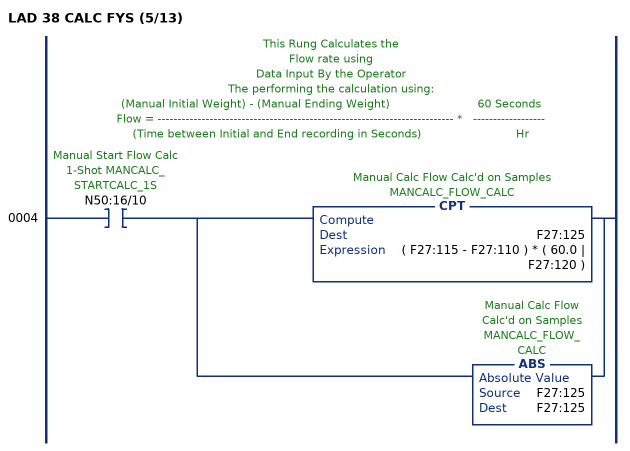
% Rung: 4 %
% This Rung Calculates the
% Flow rate using
% Data Input By the Operator
% The performing the calculation using:
% 
%              (Manual Initial Weight) - (Manual Ending Weight)                         60 Seconds
% Flow = -------------------------------------------------------------------------- *   ------------------
%    (Time between Initial and End recording in Seconds)                           Hr %
SOR XIC N50:16/10 BST CPT F27:125 " ( F27:115 - F27:110 ) * ( 60.0 | F27:120 ) " NXB ABS F27:125 F27:125 BND EOR
%   N50:16/10  MANCALC_STARTCALC_1S  "Manual Start Flow Calc 1-Shot" %
%   F27:125  MANCALC_FLOW_CALC  "Manual Calc Flow Calc'd on Samples" %
%   F27:115  MANCALC_END_VALUE  "Manual Calc End Value for Flow Calc (Lb's)" %
%   F27:110  MANCALC_INIT_VALUE  "Manual Calc Initial Value for Flow Calc (Lb's)" %
%   F27:120  MANCALC_TIME  "Manual Calc Time for Flow Calc (Min's)" %

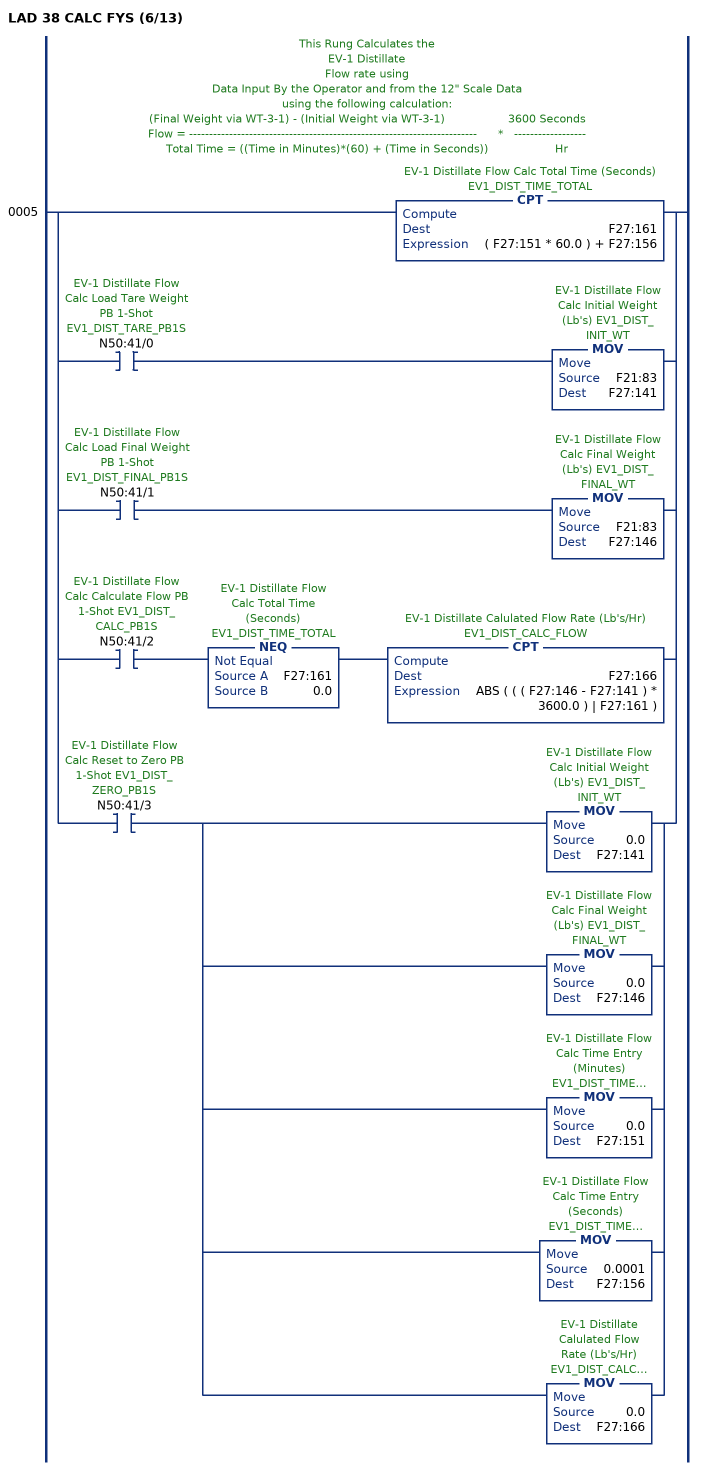
% Rung: 5 %
% This Rung Calculates the
% EV-1 Distillate
% Flow rate using
% Data Input By the Operator and from the 12" Scale Data
% using the following calculation:
% 
%              (Final Weight via WT-3-1) - (Initial Weight via WT-3-1)                  3600 Seconds
% Flow = ------------------------------------------------------------------------      *   ------------------
%    Total Time = ((Time in Minutes)*(60) + (Time in Seconds))                   Hr %
SOR BST CPT F27:161 " ( F27:151 * 60.0 ) + F27:156 " NXB XIC N50:41/0 MOV F21:83 F27:141 NXB XIC N50:41/1 MOV F21:83 F27:146 NXB XIC N50:41/2 NEQ F27:161 0.0 CPT F27:166 " ABS ( ( ( F27:146 - F27:141 ) * 3600.0 ) | F27:161 ) " NXB XIC N50:41/3 BST MOV 0.0 F27:141 NXB MOV 0.0 F27:146 NXB MOV 0.0 F27:151 NXB MOV 0.0001 F27:156 NXB MOV 0.0 F27:166 BND BND EOR
%   F27:161  EV1_DIST_TIME_TOTAL  "EV-1 Distillate Flow Calc Total Time (Seconds)" %
%   F27:151  EV1_DIST_TIME_MINS  "EV-1 Distillate Flow Calc Time Entry (Minutes)" %
%   F27:156  EV1_DIST_TIME_SECS  "EV-1 Distillate Flow Calc Time Entry (Seconds)" %
%   N50:41/0  EV1_DIST_TARE_PB1S  "EV-1 Distillate Flow Calc Load Tare Weight PB 1-Shot" %
%   F21:83  WY0301  "WY-3-1 Platform Scale No-3 Weight 12" x 12" Scale" %
%   F27:141  EV1_DIST_INIT_WT  "EV-1 Distillate Flow Calc Initial Weight (Lb's)" %
%   N50:41/1  EV1_DIST_FINAL_PB1S  "EV-1 Distillate Flow Calc Load Final Weight PB 1-Shot" %
%   F27:146  EV1_DIST_FINAL_WT  "EV-1 Distillate Flow Calc Final Weight (Lb's)" %
%   N50:41/2  EV1_DIST_CALC_PB1S  "EV-1 Distillate Flow Calc Calculate Flow PB 1-Shot" %
%   F27:166  EV1_DIST_CALC_FLOW  "EV-1 Distillate Calulated Flow Rate (Lb's/Hr)" %
%   N50:41/3  EV1_DIST_ZERO_PB1S  "EV-1 Distillate Flow Calc Reset to Zero PB 1-Shot" %

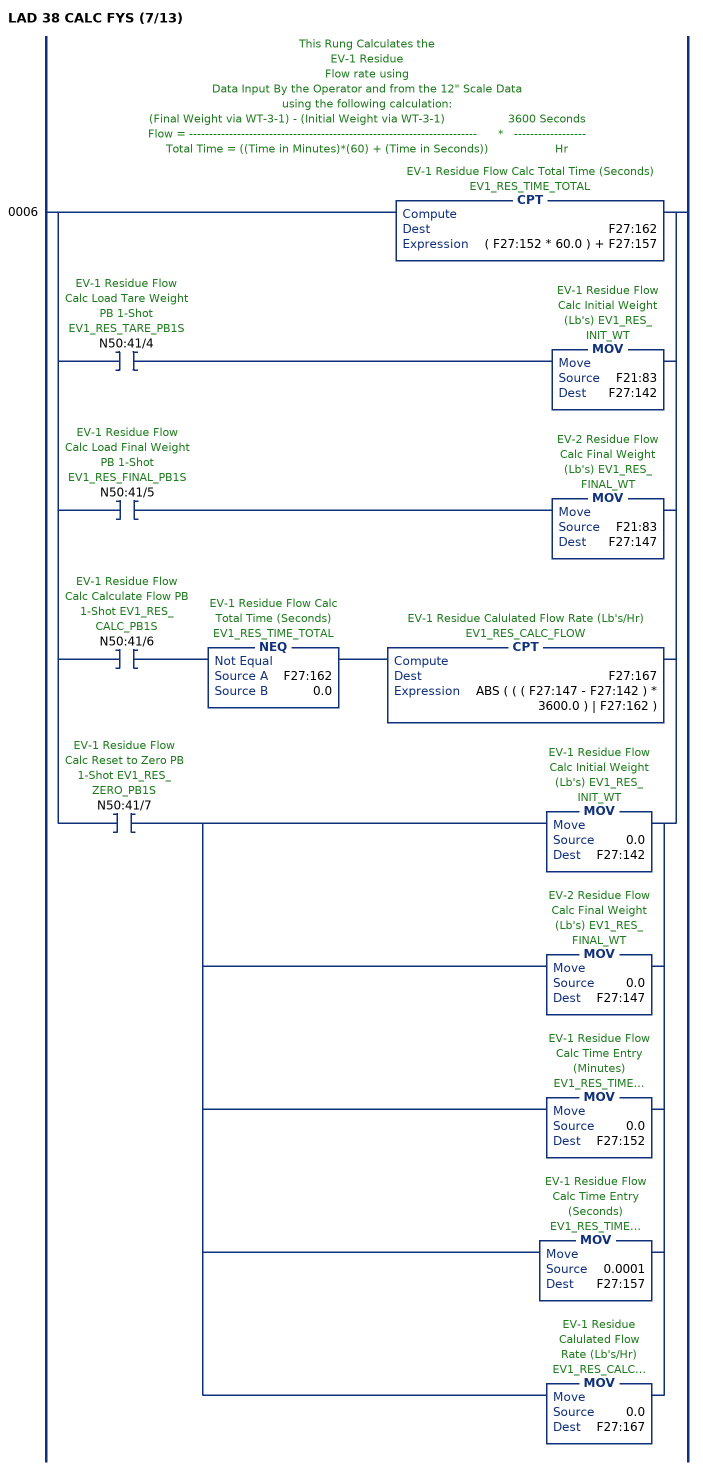
% Rung: 6 %
% This Rung Calculates the
% EV-1 Residue
% Flow rate using
% Data Input By the Operator and from the 12" Scale Data
% using the following calculation:
% 
%              (Final Weight via WT-3-1) - (Initial Weight via WT-3-1)                  3600 Seconds
% Flow = ------------------------------------------------------------------------      *   ------------------
%    Total Time = ((Time in Minutes)*(60) + (Time in Seconds))                   Hr %
SOR BST CPT F27:162 " ( F27:152 * 60.0 ) + F27:157 " NXB XIC N50:41/4 MOV F21:83 F27:142 NXB XIC N50:41/5 MOV F21:83 F27:147 NXB XIC N50:41/6 NEQ F27:162 0.0 CPT F27:167 " ABS ( ( ( F27:147 - F27:142 ) * 3600.0 ) | F27:162 ) " NXB XIC N50:41/7 BST MOV 0.0 F27:142 NXB MOV 0.0 F27:147 NXB MOV 0.0 F27:152 NXB MOV 0.0001 F27:157 NXB MOV 0.0 F27:167 BND BND EOR
%   F27:162  EV1_RES_TIME_TOTAL  "EV-1 Residue Flow Calc Total Time (Seconds)" %
%   F27:152  EV1_RES_TIME_MINS  "EV-1 Residue Flow Calc Time Entry (Minutes)" %
%   F27:157  EV1_RES_TIME_SECS  "EV-1 Residue Flow Calc Time Entry (Seconds)" %
%   N50:41/4  EV1_RES_TARE_PB1S  "EV-1 Residue Flow Calc Load Tare Weight PB 1-Shot" %
%   F21:83  WY0301  "WY-3-1 Platform Scale No-3 Weight 12" x 12" Scale" %
%   F27:142  EV1_RES_INIT_WT  "EV-1 Residue Flow Calc Initial Weight (Lb's)" %
%   N50:41/5  EV1_RES_FINAL_PB1S  "EV-1 Residue Flow Calc Load Final Weight PB 1-Shot" %
%   F27:147  EV1_RES_FINAL_WT  "EV-2 Residue Flow Calc Final Weight (Lb's)" %
%   N50:41/6  EV1_RES_CALC_PB1S  "EV-1 Residue Flow Calc Calculate Flow PB 1-Shot" %
%   F27:167  EV1_RES_CALC_FLOW  "EV-1 Residue Calulated Flow Rate (Lb's/Hr)" %
%   N50:41/7  EV1_RES_ZERO_PB1S  "EV-1 Residue Flow Calc Reset to Zero PB 1-Shot" %

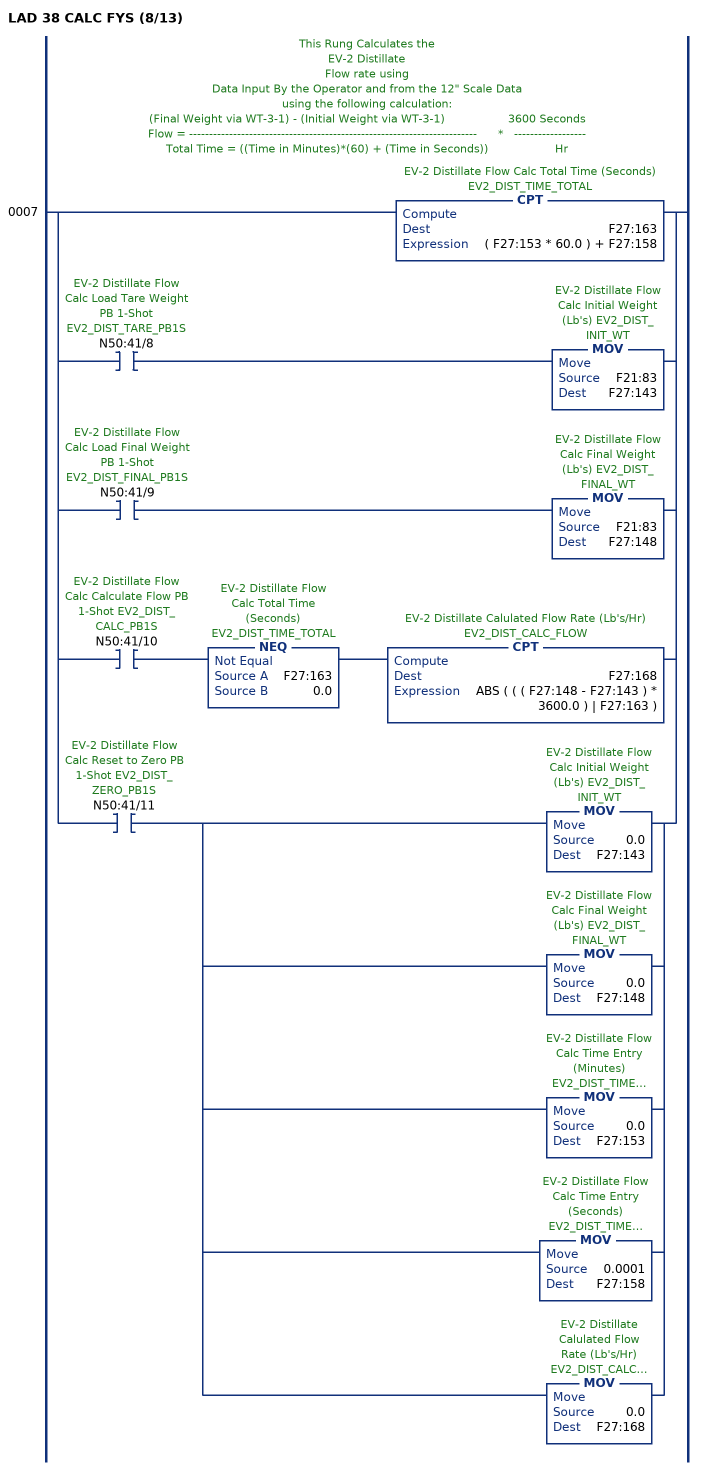
% Rung: 7 %
% This Rung Calculates the
% EV-2 Distillate
% Flow rate using
% Data Input By the Operator and from the 12" Scale Data
% using the following calculation:
% 
%              (Final Weight via WT-3-1) - (Initial Weight via WT-3-1)                  3600 Seconds
% Flow = ------------------------------------------------------------------------      *   ------------------
%    Total Time = ((Time in Minutes)*(60) + (Time in Seconds))                   Hr %
SOR BST CPT F27:163 " ( F27:153 * 60.0 ) + F27:158 " NXB XIC N50:41/8 MOV F21:83 F27:143 NXB XIC N50:41/9 MOV F21:83 F27:148 NXB XIC N50:41/10 NEQ F27:163 0.0 CPT F27:168 " ABS ( ( ( F27:148 - F27:143 ) * 3600.0 ) | F27:163 ) " NXB XIC N50:41/11 BST MOV 0.0 F27:143 NXB MOV 0.0 F27:148 NXB MOV 0.0 F27:153 NXB MOV 0.0001 F27:158 NXB MOV 0.0 F27:168 BND BND EOR
%   F27:163  EV2_DIST_TIME_TOTAL  "EV-2 Distillate Flow Calc Total Time (Seconds)" %
%   F27:153  EV2_DIST_TIME_MINS  "EV-2 Distillate Flow Calc Time Entry (Minutes)" %
%   F27:158  EV2_DIST_TIME_SECS  "EV-2 Distillate Flow Calc Time Entry (Seconds)" %
%   N50:41/8  EV2_DIST_TARE_PB1S  "EV-2 Distillate Flow Calc Load Tare Weight PB 1-Shot" %
%   F21:83  WY0301  "WY-3-1 Platform Scale No-3 Weight 12" x 12" Scale" %
%   F27:143  EV2_DIST_INIT_WT  "EV-2 Distillate Flow Calc Initial Weight (Lb's)" %
%   N50:41/9  EV2_DIST_FINAL_PB1S  "EV-2 Distillate Flow Calc Load Final Weight PB 1-Shot" %
%   F27:148  EV2_DIST_FINAL_WT  "EV-2 Distillate Flow Calc Final Weight (Lb's)" %
%   N50:41/10  EV2_DIST_CALC_PB1S  "EV-2 Distillate Flow Calc Calculate Flow PB 1-Shot" %
%   F27:168  EV2_DIST_CALC_FLOW  "EV-2 Distillate Calulated Flow Rate (Lb's/Hr)" %
%   N50:41/11  EV2_DIST_ZERO_PB1S  "EV-2 Distillate Flow Calc Reset to Zero PB 1-Shot" %

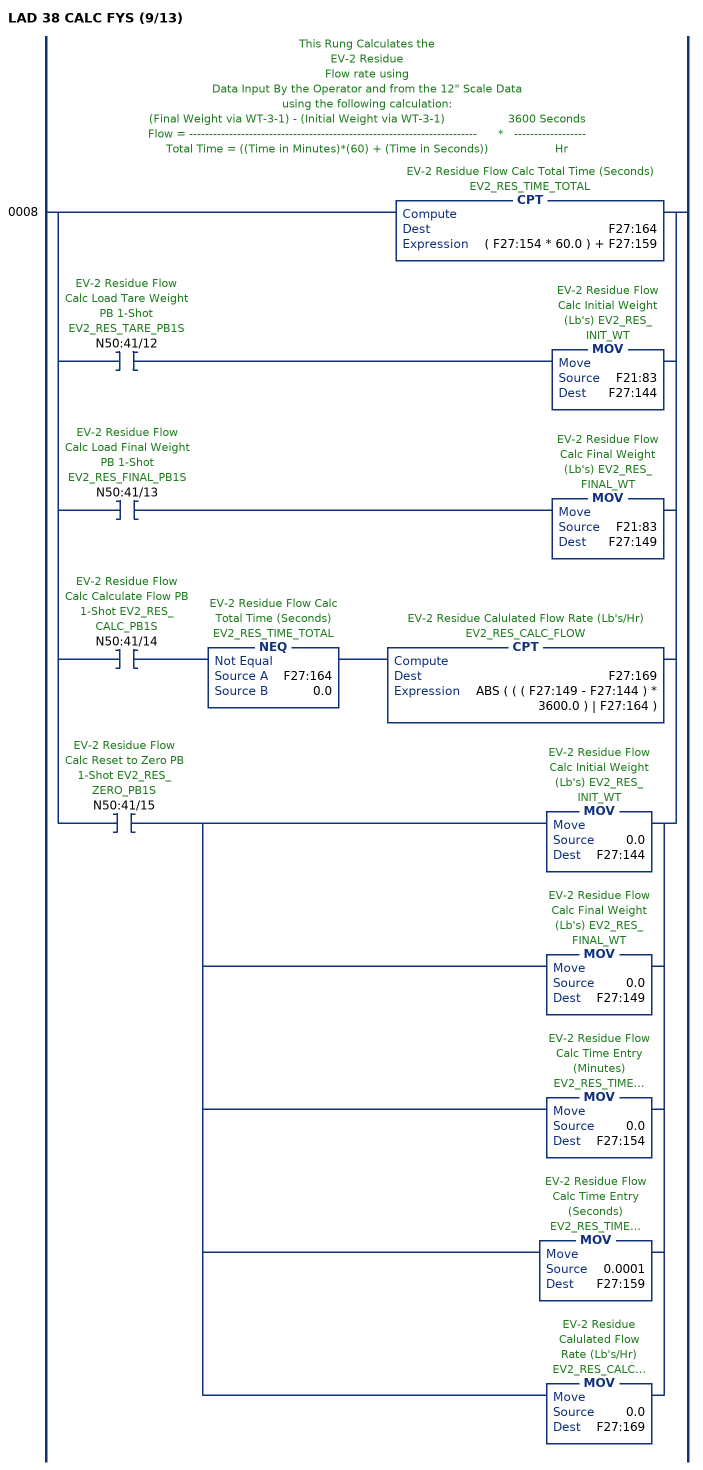
% Rung: 8 %
% This Rung Calculates the
% EV-2 Residue
% Flow rate using
% Data Input By the Operator and from the 12" Scale Data
% using the following calculation:
% 
%              (Final Weight via WT-3-1) - (Initial Weight via WT-3-1)                  3600 Seconds
% Flow = ------------------------------------------------------------------------      *   ------------------
%    Total Time = ((Time in Minutes)*(60) + (Time in Seconds))                   Hr %
SOR BST CPT F27:164 " ( F27:154 * 60.0 ) + F27:159 " NXB XIC N50:41/12 MOV F21:83 F27:144 NXB XIC N50:41/13 MOV F21:83 F27:149 NXB XIC N50:41/14 NEQ F27:164 0.0 CPT F27:169 " ABS ( ( ( F27:149 - F27:144 ) * 3600.0 ) | F27:164 ) " NXB XIC N50:41/15 BST MOV 0.0 F27:144 NXB MOV 0.0 F27:149 NXB MOV 0.0 F27:154 NXB MOV 0.0001 F27:159 NXB MOV 0.0 F27:169 BND BND EOR
%   F27:164  EV2_RES_TIME_TOTAL  "EV-2 Residue Flow Calc Total Time (Seconds)" %
%   F27:154  EV2_RES_TIME_MINS  "EV-2 Residue Flow Calc Time Entry (Minutes)" %
%   F27:159  EV2_RES_TIME_SECS  "EV-2 Residue Flow Calc Time Entry (Seconds)" %
%   N50:41/12  EV2_RES_TARE_PB1S  "EV-2 Residue Flow Calc Load Tare Weight PB 1-Shot" %
%   F21:83  WY0301  "WY-3-1 Platform Scale No-3 Weight 12" x 12" Scale" %
%   F27:144  EV2_RES_INIT_WT  "EV-2 Residue Flow Calc Initial Weight (Lb's)" %
%   N50:41/13  EV2_RES_FINAL_PB1S  "EV-2 Residue Flow Calc Load Final Weight PB 1-Shot" %
%   F27:149  EV2_RES_FINAL_WT  "EV-2 Residue Flow Calc Final Weight (Lb's)" %
%   N50:41/14  EV2_RES_CALC_PB1S  "EV-2 Residue Flow Calc Calculate Flow PB 1-Shot" %
%   F27:169  EV2_RES_CALC_FLOW  "EV-2 Residue Calulated Flow Rate (Lb's/Hr)" %
%   N50:41/15  EV2_RES_ZERO_PB1S  "EV-2 Residue Flow Calc Reset to Zero PB 1-Shot" %

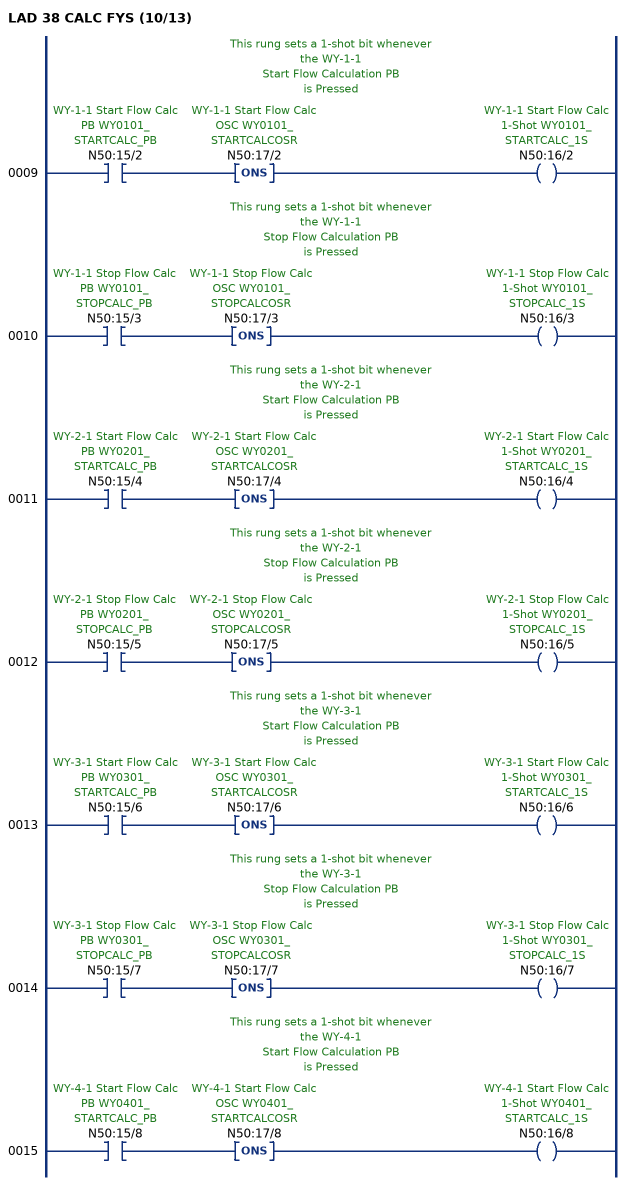
% Rung: 9 %
% This rung sets a 1-shot bit whenever
% the WY-1-1
% Start Flow Calculation PB
% is Pressed %
SOR XIC N50:15/2 OSR N50:17/2 OTE N50:16/2 EOR
%   N50:15/2  WY0101_STARTCALC_PB  "WY-1-1 Start Flow Calc PB" %
%   N50:17/2  WY0101_STARTCALCOSR  "WY-1-1 Start Flow Calc OSC" %
%   N50:16/2  WY0101_STARTCALC_1S  "WY-1-1 Start Flow Calc 1-Shot" %
% Rung: 10 %
% This rung sets a 1-shot bit whenever
% the WY-1-1
% Stop Flow Calculation PB
% is Pressed %
SOR XIC N50:15/3 OSR N50:17/3 OTE N50:16/3 EOR
%   N50:15/3  WY0101_STOPCALC_PB  "WY-1-1 Stop Flow Calc PB" %
%   N50:17/3  WY0101_STOPCALCOSR  "WY-1-1 Stop Flow Calc OSC" %
%   N50:16/3  WY0101_STOPCALC_1S  "WY-1-1 Stop Flow Calc 1-Shot" %
% Rung: 11 %
% This rung sets a 1-shot bit whenever
% the WY-2-1
% Start Flow Calculation PB
% is Pressed %
SOR XIC N50:15/4 OSR N50:17/4 OTE N50:16/4 EOR
%   N50:15/4  WY0201_STARTCALC_PB  "WY-2-1 Start Flow Calc PB" %
%   N50:17/4  WY0201_STARTCALCOSR  "WY-2-1 Start Flow Calc OSC" %
%   N50:16/4  WY0201_STARTCALC_1S  "WY-2-1 Start Flow Calc 1-Shot" %
% Rung: 12 %
% This rung sets a 1-shot bit whenever
% the WY-2-1
% Stop Flow Calculation PB
% is Pressed %
SOR XIC N50:15/5 OSR N50:17/5 OTE N50:16/5 EOR
%   N50:15/5  WY0201_STOPCALC_PB  "WY-2-1 Stop Flow Calc PB" %
%   N50:17/5  WY0201_STOPCALCOSR  "WY-2-1 Stop Flow Calc OSC" %
%   N50:16/5  WY0201_STOPCALC_1S  "WY-2-1 Stop Flow Calc 1-Shot" %
% Rung: 13 %
% This rung sets a 1-shot bit whenever
% the WY-3-1
% Start Flow Calculation PB
% is Pressed %
SOR XIC N50:15/6 OSR N50:17/6 OTE N50:16/6 EOR
%   N50:15/6  WY0301_STARTCALC_PB  "WY-3-1 Start Flow Calc PB" %
%   N50:17/6  WY0301_STARTCALCOSR  "WY-3-1 Start Flow Calc OSC" %
%   N50:16/6  WY0301_STARTCALC_1S  "WY-3-1 Start Flow Calc 1-Shot" %
% Rung: 14 %
% This rung sets a 1-shot bit whenever
% the WY-3-1
% Stop Flow Calculation PB
% is Pressed %
SOR XIC N50:15/7 OSR N50:17/7 OTE N50:16/7 EOR
%   N50:15/7  WY0301_STOPCALC_PB  "WY-3-1 Stop Flow Calc PB" %
%   N50:17/7  WY0301_STOPCALCOSR  "WY-3-1 Stop Flow Calc OSC" %
%   N50:16/7  WY0301_STOPCALC_1S  "WY-3-1 Stop Flow Calc 1-Shot" %
% Rung: 15 %
% This rung sets a 1-shot bit whenever
% the WY-4-1
% Start Flow Calculation PB
% is Pressed %
SOR XIC N50:15/8 OSR N50:17/8 OTE N50:16/8 EOR
%   N50:15/8  WY0401_STARTCALC_PB  "WY-4-1 Start Flow Calc PB" %
%   N50:17/8  WY0401_STARTCALCOSR  "WY-4-1 Start Flow Calc OSC" %
%   N50:16/8  WY0401_STARTCALC_1S  "WY-4-1 Start Flow Calc 1-Shot" %

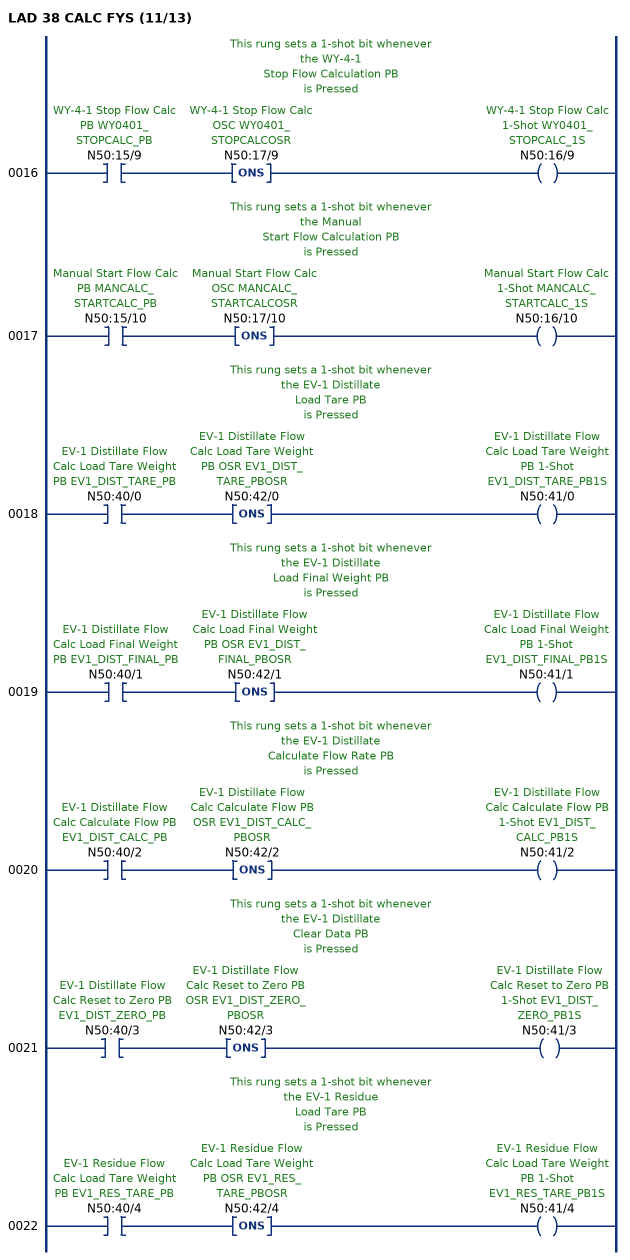
% Rung: 16 %
% This rung sets a 1-shot bit whenever
% the WY-4-1
% Stop Flow Calculation PB
% is Pressed %
SOR XIC N50:15/9 OSR N50:17/9 OTE N50:16/9 EOR
%   N50:15/9  WY0401_STOPCALC_PB  "WY-4-1 Stop Flow Calc PB" %
%   N50:17/9  WY0401_STOPCALCOSR  "WY-4-1 Stop Flow Calc OSC" %
%   N50:16/9  WY0401_STOPCALC_1S  "WY-4-1 Stop Flow Calc 1-Shot" %
% Rung: 17 %
% This rung sets a 1-shot bit whenever
% the Manual
% Start Flow Calculation PB
% is Pressed %
SOR XIC N50:15/10 OSR N50:17/10 OTE N50:16/10 EOR
%   N50:15/10  MANCALC_STARTCALC_PB  "Manual Start Flow Calc PB" %
%   N50:17/10  MANCALC_STARTCALCOSR  "Manual Start Flow Calc OSC" %
%   N50:16/10  MANCALC_STARTCALC_1S  "Manual Start Flow Calc 1-Shot" %
% Rung: 18 %
% This rung sets a 1-shot bit whenever
% the EV-1 Distillate
% Load Tare PB
% is Pressed %
SOR XIC N50:40/0 OSR N50:42/0 OTE N50:41/0 EOR
%   N50:40/0  EV1_DIST_TARE_PB  "EV-1 Distillate Flow Calc Load Tare Weight PB" %
%   N50:42/0  EV1_DIST_TARE_PBOSR  "EV-1 Distillate Flow Calc Load Tare Weight PB OSR" %
%   N50:41/0  EV1_DIST_TARE_PB1S  "EV-1 Distillate Flow Calc Load Tare Weight PB 1-Shot" %
% Rung: 19 %
% This rung sets a 1-shot bit whenever
% the EV-1 Distillate
% Load Final Weight PB
% is Pressed %
SOR XIC N50:40/1 OSR N50:42/1 OTE N50:41/1 EOR
%   N50:40/1  EV1_DIST_FINAL_PB  "EV-1 Distillate Flow Calc Load Final Weight PB" %
%   N50:42/1  EV1_DIST_FINAL_PBOSR  "EV-1 Distillate Flow Calc Load Final Weight PB OSR" %
%   N50:41/1  EV1_DIST_FINAL_PB1S  "EV-1 Distillate Flow Calc Load Final Weight PB 1-Shot" %
% Rung: 20 %
% This rung sets a 1-shot bit whenever
% the EV-1 Distillate
% Calculate Flow Rate PB
% is Pressed %
SOR XIC N50:40/2 OSR N50:42/2 OTE N50:41/2 EOR
%   N50:40/2  EV1_DIST_CALC_PB  "EV-1 Distillate Flow Calc Calculate Flow PB" %
%   N50:42/2  EV1_DIST_CALC_PBOSR  "EV-1 Distillate Flow Calc Calculate Flow PB OSR" %
%   N50:41/2  EV1_DIST_CALC_PB1S  "EV-1 Distillate Flow Calc Calculate Flow PB 1-Shot" %
% Rung: 21 %
% This rung sets a 1-shot bit whenever
% the EV-1 Distillate
% Clear Data PB
% is Pressed %
SOR XIC N50:40/3 OSR N50:42/3 OTE N50:41/3 EOR
%   N50:40/3  EV1_DIST_ZERO_PB  "EV-1 Distillate Flow Calc Reset to Zero PB" %
%   N50:42/3  EV1_DIST_ZERO_PBOSR  "EV-1 Distillate Flow Calc Reset to Zero PB OSR" %
%   N50:41/3  EV1_DIST_ZERO_PB1S  "EV-1 Distillate Flow Calc Reset to Zero PB 1-Shot" %
% Rung: 22 %
% This rung sets a 1-shot bit whenever
% the EV-1 Residue
% Load Tare PB
% is Pressed %
SOR XIC N50:40/4 OSR N50:42/4 OTE N50:41/4 EOR
%   N50:40/4  EV1_RES_TARE_PB  "EV-1 Residue Flow Calc Load Tare Weight PB" %
%   N50:42/4  EV1_RES_TARE_PBOSR  "EV-1 Residue Flow Calc Load Tare Weight PB OSR" %
%   N50:41/4  EV1_RES_TARE_PB1S  "EV-1 Residue Flow Calc Load Tare Weight PB 1-Shot" %

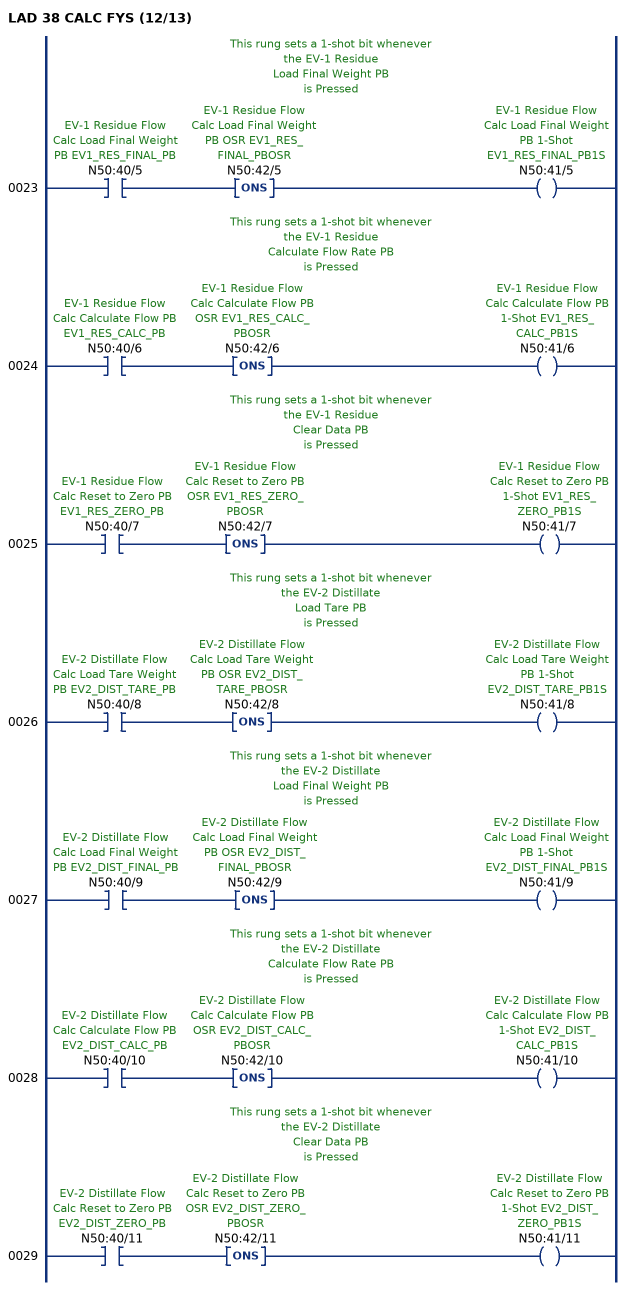
% Rung: 23 %
% This rung sets a 1-shot bit whenever
% the EV-1 Residue
% Load Final Weight PB
% is Pressed %
SOR XIC N50:40/5 OSR N50:42/5 OTE N50:41/5 EOR
%   N50:40/5  EV1_RES_FINAL_PB  "EV-1 Residue Flow Calc Load Final Weight PB" %
%   N50:42/5  EV1_RES_FINAL_PBOSR  "EV-1 Residue Flow Calc Load Final Weight PB OSR" %
%   N50:41/5  EV1_RES_FINAL_PB1S  "EV-1 Residue Flow Calc Load Final Weight PB 1-Shot" %
% Rung: 24 %
% This rung sets a 1-shot bit whenever
% the EV-1 Residue
% Calculate Flow Rate PB
% is Pressed %
SOR XIC N50:40/6 OSR N50:42/6 OTE N50:41/6 EOR
%   N50:40/6  EV1_RES_CALC_PB  "EV-1 Residue Flow Calc Calculate Flow PB" %
%   N50:42/6  EV1_RES_CALC_PBOSR  "EV-1 Residue Flow Calc Calculate Flow PB OSR" %
%   N50:41/6  EV1_RES_CALC_PB1S  "EV-1 Residue Flow Calc Calculate Flow PB 1-Shot" %
% Rung: 25 %
% This rung sets a 1-shot bit whenever
% the EV-1 Residue
% Clear Data PB
% is Pressed %
SOR XIC N50:40/7 OSR N50:42/7 OTE N50:41/7 EOR
%   N50:40/7  EV1_RES_ZERO_PB  "EV-1 Residue Flow Calc Reset to Zero PB" %
%   N50:42/7  EV1_RES_ZERO_PBOSR  "EV-1 Residue Flow Calc Reset to Zero PB OSR" %
%   N50:41/7  EV1_RES_ZERO_PB1S  "EV-1 Residue Flow Calc Reset to Zero PB 1-Shot" %
% Rung: 26 %
% This rung sets a 1-shot bit whenever
% the EV-2 Distillate
% Load Tare PB
% is Pressed %
SOR XIC N50:40/8 OSR N50:42/8 OTE N50:41/8 EOR
%   N50:40/8  EV2_DIST_TARE_PB  "EV-2 Distillate Flow Calc Load Tare Weight PB" %
%   N50:42/8  EV2_DIST_TARE_PBOSR  "EV-2 Distillate Flow Calc Load Tare Weight PB OSR" %
%   N50:41/8  EV2_DIST_TARE_PB1S  "EV-2 Distillate Flow Calc Load Tare Weight PB 1-Shot" %
% Rung: 27 %
% This rung sets a 1-shot bit whenever
% the EV-2 Distillate
% Load Final Weight PB
% is Pressed %
SOR XIC N50:40/9 OSR N50:42/9 OTE N50:41/9 EOR
%   N50:40/9  EV2_DIST_FINAL_PB  "EV-2 Distillate Flow Calc Load Final Weight PB" %
%   N50:42/9  EV2_DIST_FINAL_PBOSR  "EV-2 Distillate Flow Calc Load Final Weight PB OSR" %
%   N50:41/9  EV2_DIST_FINAL_PB1S  "EV-2 Distillate Flow Calc Load Final Weight PB 1-Shot" %
% Rung: 28 %
% This rung sets a 1-shot bit whenever
% the EV-2 Distillate
% Calculate Flow Rate PB
% is Pressed %
SOR XIC N50:40/10 OSR N50:42/10 OTE N50:41/10 EOR
%   N50:40/10  EV2_DIST_CALC_PB  "EV-2 Distillate Flow Calc Calculate Flow PB" %
%   N50:42/10  EV2_DIST_CALC_PBOSR  "EV-2 Distillate Flow Calc Calculate Flow PB OSR" %
%   N50:41/10  EV2_DIST_CALC_PB1S  "EV-2 Distillate Flow Calc Calculate Flow PB 1-Shot" %
% Rung: 29 %
% This rung sets a 1-shot bit whenever
% the EV-2 Distillate
% Clear Data PB
% is Pressed %
SOR XIC N50:40/11 OSR N50:42/11 OTE N50:41/11 EOR
%   N50:40/11  EV2_DIST_ZERO_PB  "EV-2 Distillate Flow Calc Reset to Zero PB" %
%   N50:42/11  EV2_DIST_ZERO_PBOSR  "EV-2 Distillate Flow Calc Reset to Zero PB OSR" %
%   N50:41/11  EV2_DIST_ZERO_PB1S  "EV-2 Distillate Flow Calc Reset to Zero PB 1-Shot" %

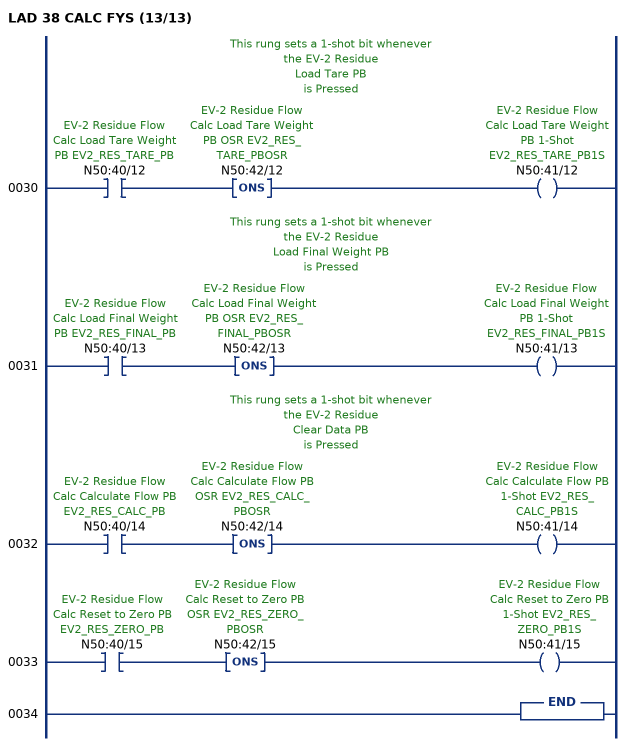
% Rung: 30 %
% This rung sets a 1-shot bit whenever
% the EV-2 Residue
% Load Tare PB
% is Pressed %
SOR XIC N50:40/12 OSR N50:42/12 OTE N50:41/12 EOR
%   N50:40/12  EV2_RES_TARE_PB  "EV-2 Residue Flow Calc Load Tare Weight PB" %
%   N50:42/12  EV2_RES_TARE_PBOSR  "EV-2 Residue Flow Calc Load Tare Weight PB OSR" %
%   N50:41/12  EV2_RES_TARE_PB1S  "EV-2 Residue Flow Calc Load Tare Weight PB 1-Shot" %
% Rung: 31 %
% This rung sets a 1-shot bit whenever
% the EV-2 Residue
% Load Final Weight PB
% is Pressed %
SOR XIC N50:40/13 OSR N50:42/13 OTE N50:41/13 EOR
%   N50:40/13  EV2_RES_FINAL_PB  "EV-2 Residue Flow Calc Load Final Weight PB" %
%   N50:42/13  EV2_RES_FINAL_PBOSR  "EV-2 Residue Flow Calc Load Final Weight PB OSR" %
%   N50:41/13  EV2_RES_FINAL_PB1S  "EV-2 Residue Flow Calc Load Final Weight PB 1-Shot" %
% Rung: 32 %
% This rung sets a 1-shot bit whenever
% the EV-2 Residue
% Clear Data PB
% is Pressed %
SOR XIC N50:40/14 OSR N50:42/14 OTE N50:41/14 EOR
%   N50:40/14  EV2_RES_CALC_PB  "EV-2 Residue Flow Calc Calculate Flow PB" %
%   N50:42/14  EV2_RES_CALC_PBOSR  "EV-2 Residue Flow Calc Calculate Flow PB OSR" %
%   N50:41/14  EV2_RES_CALC_PB1S  "EV-2 Residue Flow Calc Calculate Flow PB 1-Shot" %
% Rung: 33 %
SOR XIC N50:40/15 OSR N50:42/15 OTE N50:41/15 EOR
%   N50:40/15  EV2_RES_ZERO_PB  "EV-2 Residue Flow Calc Reset to Zero PB" %
%   N50:42/15  EV2_RES_ZERO_PBOSR  "EV-2 Residue Flow Calc Reset to Zero PB OSR" %
%   N50:41/15  EV2_RES_ZERO_PB1S  "EV-2 Residue Flow Calc Reset to Zero PB 1-Shot" %
% Rung: 34 %
SOR END EOR

LADDER 39 "CALC ITS"    % Calculate SY Current Values %
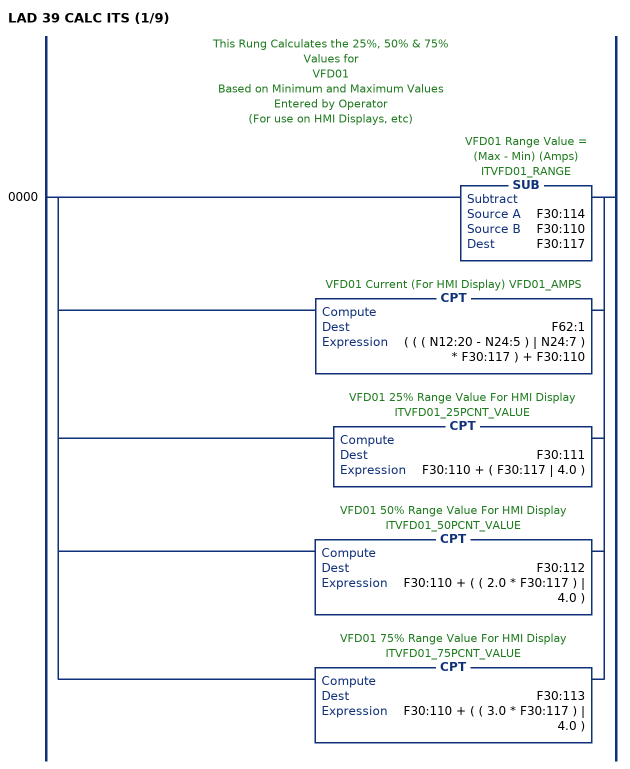
% Rung: 0 %
% This Rung Calculates the 25%, 50% & 75%
% Values for
% VFD01
% Based on Minimum and Maximum Values
% Entered by Operator
% (For use on HMI Displays, etc) %
SOR BST SUB F30:114 F30:110 F30:117 NXB CPT F62:1 " ( ( ( N12:20 - N24:5 ) | N24:7 ) * F30:117 ) + F30:110 " NXB CPT F30:111 " F30:110 + ( F30:117 | 4.0 ) " NXB CPT F30:112 " F30:110 + ( ( 2.0 * F30:117 ) | 4.0 ) " NXB CPT F30:113 " F30:110 + ( ( 3.0 * F30:117 ) | 4.0 ) " BND EOR
%   F30:114  ITVFD01_MAX  "VFD01 Maximum Value (Amps)" %
%   F30:110  ITVFD01_MIN  "VFD01 Minimum Value (Amps)" %
%   F30:117  ITVFD01_RANGE  "VFD01 Range Value = (Max - Min) (Amps)" %
%   F62:1  VFD01_AMPS  "VFD01 Current (For HMI Display)" %
%   N12:20  VFD01_BIN_AMPS  "VFD01 Binary Amps" %
%   N24:5  AI_VOLTAGE_MIN  "Analog Input Minimum Value = 0 VDC (From AI Module)" %
%   N24:7  AI_VOLTAGE_RANGE  "Analog Input Voltage Range Value = (AI_MAX - AI_MIN) For Use Elswhere" %
%   F30:111  ITVFD01_25PCNT_VALUE  "VFD01 25% Range Value For HMI Display" %
%   F30:112  ITVFD01_50PCNT_VALUE  "VFD01 50% Range Value For HMI Display" %
%   F30:113  ITVFD01_75PCNT_VALUE  "VFD01 75% Range Value For HMI Display" %

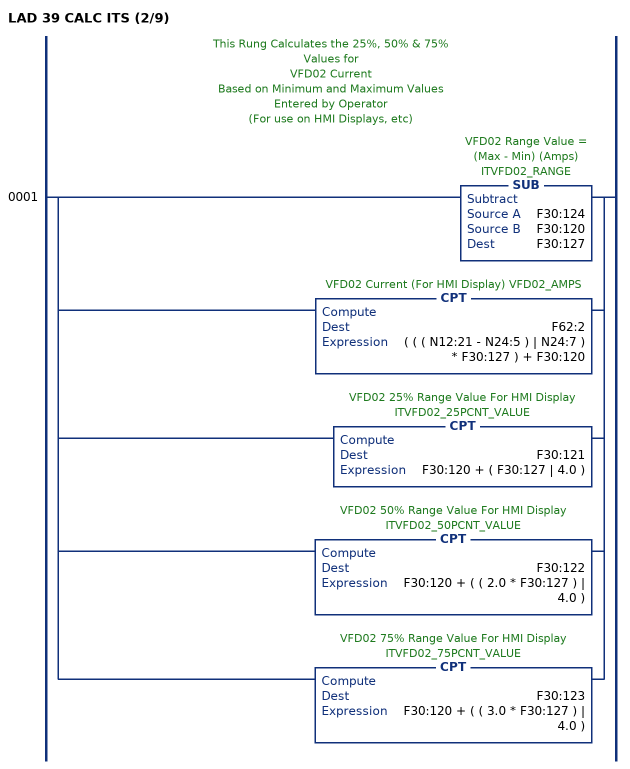
% Rung: 1 %
% This Rung Calculates the 25%, 50% & 75%
% Values for
% VFD02 Current
% Based on Minimum and Maximum Values
% Entered by Operator
% (For use on HMI Displays, etc) %
SOR BST SUB F30:124 F30:120 F30:127 NXB CPT F62:2 " ( ( ( N12:21 - N24:5 ) | N24:7 ) * F30:127 ) + F30:120 " NXB CPT F30:121 " F30:120 + ( F30:127 | 4.0 ) " NXB CPT F30:122 " F30:120 + ( ( 2.0 * F30:127 ) | 4.0 ) " NXB CPT F30:123 " F30:120 + ( ( 3.0 * F30:127 ) | 4.0 ) " BND EOR
%   F30:124  ITVFD02_MAX  "VFD02 Maximum Value (Amps)" %
%   F30:120  ITVFD02_MIN  "VFD02 Minimum Value (Amps)" %
%   F30:127  ITVFD02_RANGE  "VFD02 Range Value = (Max - Min) (Amps)" %
%   F62:2  VFD02_AMPS  "VFD02 Current (For HMI Display)" %
%   N12:21  VFD02_BIN_AMPS  "VFD02 Binary Amps" %
%   N24:5  AI_VOLTAGE_MIN  "Analog Input Minimum Value = 0 VDC (From AI Module)" %
%   N24:7  AI_VOLTAGE_RANGE  "Analog Input Voltage Range Value = (AI_MAX - AI_MIN) For Use Elswhere" %
%   F30:121  ITVFD02_25PCNT_VALUE  "VFD02 25% Range Value For HMI Display" %
%   F30:122  ITVFD02_50PCNT_VALUE  "VFD02 50% Range Value For HMI Display" %
%   F30:123  ITVFD02_75PCNT_VALUE  "VFD02 75% Range Value For HMI Display" %

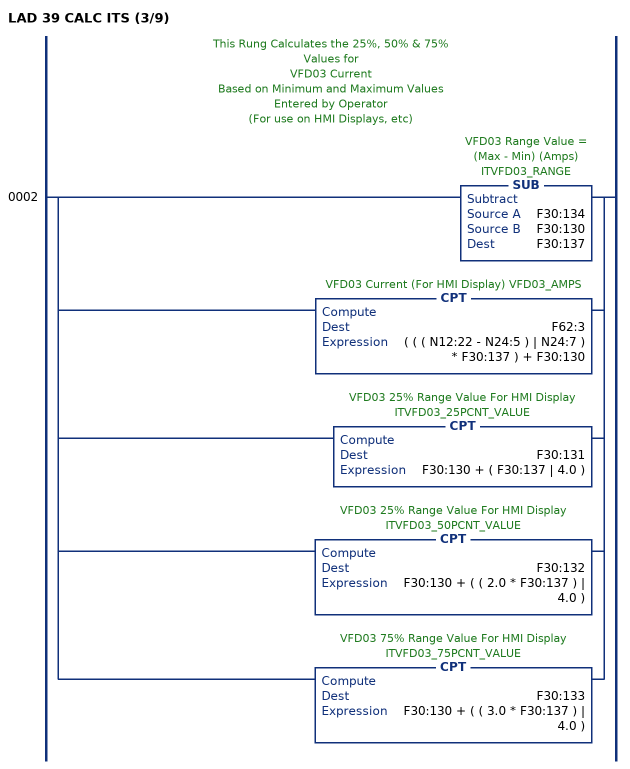
% Rung: 2 %
% This Rung Calculates the 25%, 50% & 75%
% Values for
% VFD03 Current
% Based on Minimum and Maximum Values
% Entered by Operator
% (For use on HMI Displays, etc) %
SOR BST SUB F30:134 F30:130 F30:137 NXB CPT F62:3 " ( ( ( N12:22 - N24:5 ) | N24:7 ) * F30:137 ) + F30:130 " NXB CPT F30:131 " F30:130 + ( F30:137 | 4.0 ) " NXB CPT F30:132 " F30:130 + ( ( 2.0 * F30:137 ) | 4.0 ) " NXB CPT F30:133 " F30:130 + ( ( 3.0 * F30:137 ) | 4.0 ) " BND EOR
%   F30:134  ITVFD03_MAX  "VFD03 Maximum Value (Amps)" %
%   F30:130  ITVFD03_MIN  "VFD03 Minimum Value (Amps)" %
%   F30:137  ITVFD03_RANGE  "VFD03 Range Value = (Max - Min) (Amps)" %
%   F62:3  VFD03_AMPS  "VFD03 Current (For HMI Display)" %
%   N12:22  VFD03_BIN_AMPS  "VFD03 Binary Amps" %
%   N24:5  AI_VOLTAGE_MIN  "Analog Input Minimum Value = 0 VDC (From AI Module)" %
%   N24:7  AI_VOLTAGE_RANGE  "Analog Input Voltage Range Value = (AI_MAX - AI_MIN) For Use Elswhere" %
%   F30:131  ITVFD03_25PCNT_VALUE  "VFD03 25% Range Value For HMI Display" %
%   F30:132  ITVFD03_50PCNT_VALUE  "VFD03 25% Range Value For HMI Display" %
%   F30:133  ITVFD03_75PCNT_VALUE  "VFD03 75% Range Value For HMI Display" %

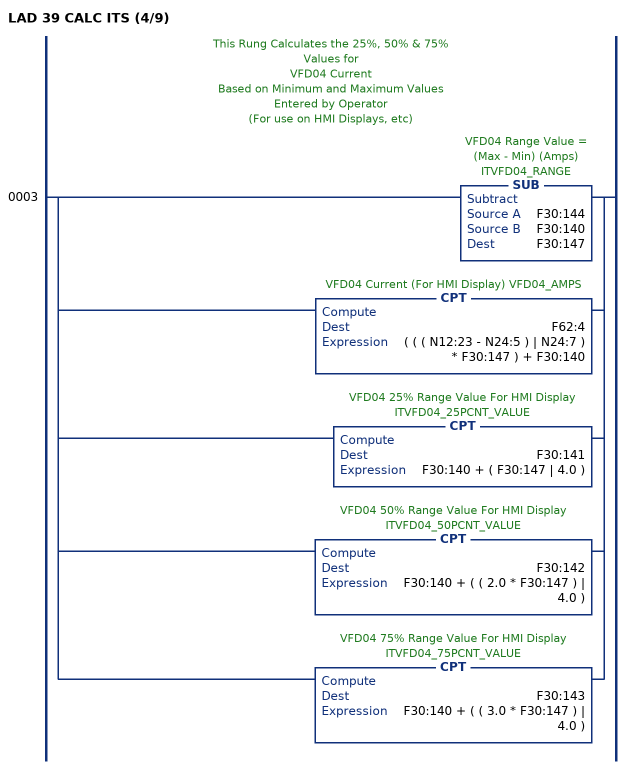
% Rung: 3 %
% This Rung Calculates the 25%, 50% & 75%
% Values for
% VFD04 Current
% Based on Minimum and Maximum Values
% Entered by Operator
% (For use on HMI Displays, etc) %
SOR BST SUB F30:144 F30:140 F30:147 NXB CPT F62:4 " ( ( ( N12:23 - N24:5 ) | N24:7 ) * F30:147 ) + F30:140 " NXB CPT F30:141 " F30:140 + ( F30:147 | 4.0 ) " NXB CPT F30:142 " F30:140 + ( ( 2.0 * F30:147 ) | 4.0 ) " NXB CPT F30:143 " F30:140 + ( ( 3.0 * F30:147 ) | 4.0 ) " BND EOR
%   F30:144  ITVFD04_MAX  "VFD04 Maximum Value (Amps)" %
%   F30:140  ITVFD04_MIN  "VFD04 Minimum Value (Amps)" %
%   F30:147  ITVFD04_RANGE  "VFD04 Range Value = (Max - Min) (Amps)" %
%   F62:4  VFD04_AMPS  "VFD04 Current (For HMI Display)" %
%   N12:23  VFD04_BIN_AMPS  "VFD04 Binary Amps" %
%   N24:5  AI_VOLTAGE_MIN  "Analog Input Minimum Value = 0 VDC (From AI Module)" %
%   N24:7  AI_VOLTAGE_RANGE  "Analog Input Voltage Range Value = (AI_MAX - AI_MIN) For Use Elswhere" %
%   F30:141  ITVFD04_25PCNT_VALUE  "VFD04 25% Range Value For HMI Display" %
%   F30:142  ITVFD04_50PCNT_VALUE  "VFD04 50% Range Value For HMI Display" %
%   F30:143  ITVFD04_75PCNT_VALUE  "VFD04 75% Range Value For HMI Display" %

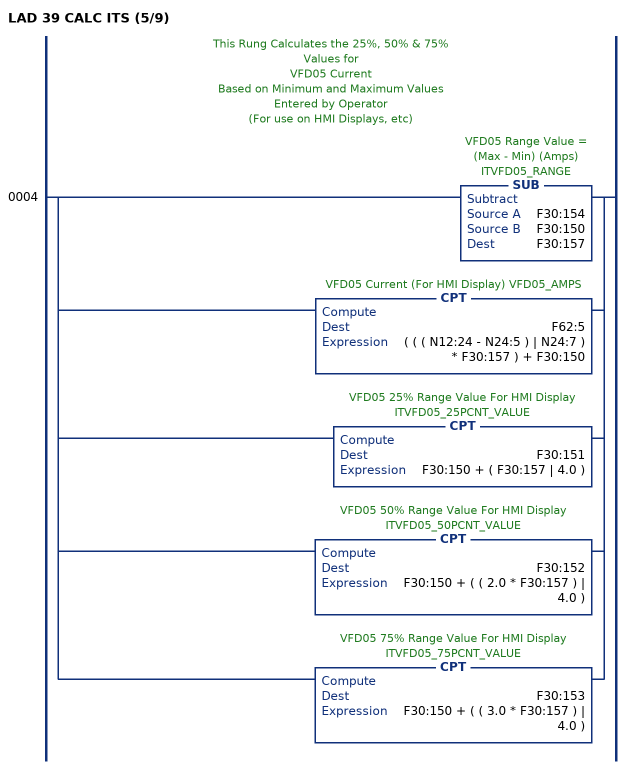
% Rung: 4 %
% This Rung Calculates the 25%, 50% & 75%
% Values for
% VFD05 Current
% Based on Minimum and Maximum Values
% Entered by Operator
% (For use on HMI Displays, etc) %
SOR BST SUB F30:154 F30:150 F30:157 NXB CPT F62:5 " ( ( ( N12:24 - N24:5 ) | N24:7 ) * F30:157 ) + F30:150 " NXB CPT F30:151 " F30:150 + ( F30:157 | 4.0 ) " NXB CPT F30:152 " F30:150 + ( ( 2.0 * F30:157 ) | 4.0 ) " NXB CPT F30:153 " F30:150 + ( ( 3.0 * F30:157 ) | 4.0 ) " BND EOR
%   F30:154  ITVFD05_MAX  "VFD05 Maximum Value (Amps)" %
%   F30:150  ITVFD05_MIN  "VFD05 Minimum Value (Amps)" %
%   F30:157  ITVFD05_RANGE  "VFD05 Range Value = (Max - Min) (Amps)" %
%   F62:5  VFD05_AMPS  "VFD05 Current (For HMI Display)" %
%   N12:24  VFD05_BIN_AMPS  "VFD05 Binary Amps" %
%   N24:5  AI_VOLTAGE_MIN  "Analog Input Minimum Value = 0 VDC (From AI Module)" %
%   N24:7  AI_VOLTAGE_RANGE  "Analog Input Voltage Range Value = (AI_MAX - AI_MIN) For Use Elswhere" %
%   F30:151  ITVFD05_25PCNT_VALUE  "VFD05 25% Range Value For HMI Display" %
%   F30:152  ITVFD05_50PCNT_VALUE  "VFD05 50% Range Value For HMI Display" %
%   F30:153  ITVFD05_75PCNT_VALUE  "VFD05 75% Range Value For HMI Display" %

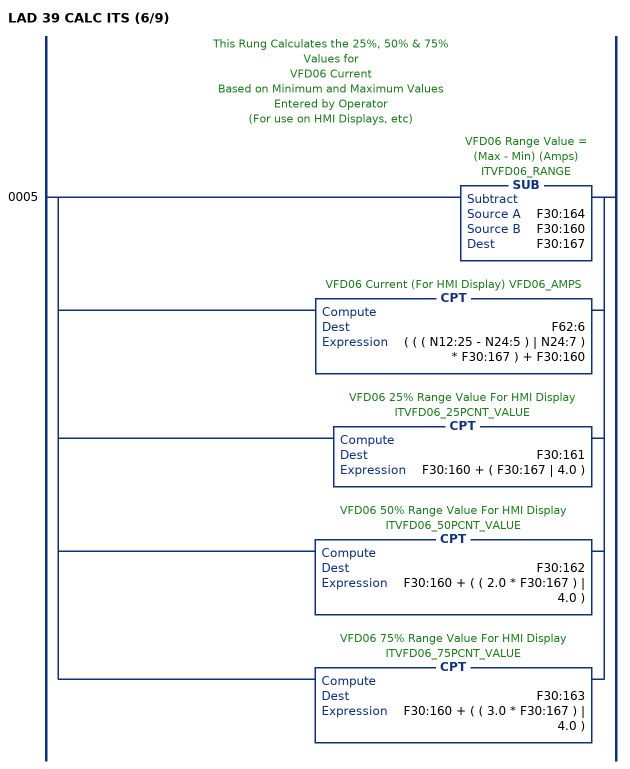
% Rung: 5 %
% This Rung Calculates the 25%, 50% & 75%
% Values for
% VFD06 Current
% Based on Minimum and Maximum Values
% Entered by Operator
% (For use on HMI Displays, etc) %
SOR BST SUB F30:164 F30:160 F30:167 NXB CPT F62:6 " ( ( ( N12:25 - N24:5 ) | N24:7 ) * F30:167 ) + F30:160 " NXB CPT F30:161 " F30:160 + ( F30:167 | 4.0 ) " NXB CPT F30:162 " F30:160 + ( ( 2.0 * F30:167 ) | 4.0 ) " NXB CPT F30:163 " F30:160 + ( ( 3.0 * F30:167 ) | 4.0 ) " BND EOR
%   F30:164  ITVFD06_MAX  "VFD06 Maximum Value (Amps)" %
%   F30:160  ITVFD06_MIN  "VFD06 Minimum Value (Amps)" %
%   F30:167  ITVFD06_RANGE  "VFD06 Range Value = (Max - Min) (Amps)" %
%   F62:6  VFD06_AMPS  "VFD06 Current (For HMI Display)" %
%   N12:25  VFD06_BIN_AMPS  "VFD06 Binary Amps" %
%   N24:5  AI_VOLTAGE_MIN  "Analog Input Minimum Value = 0 VDC (From AI Module)" %
%   N24:7  AI_VOLTAGE_RANGE  "Analog Input Voltage Range Value = (AI_MAX - AI_MIN) For Use Elswhere" %
%   F30:161  ITVFD06_25PCNT_VALUE  "VFD06 25% Range Value For HMI Display" %
%   F30:162  ITVFD06_50PCNT_VALUE  "VFD06 50% Range Value For HMI Display" %
%   F30:163  ITVFD06_75PCNT_VALUE  "VFD06 75% Range Value For HMI Display" %

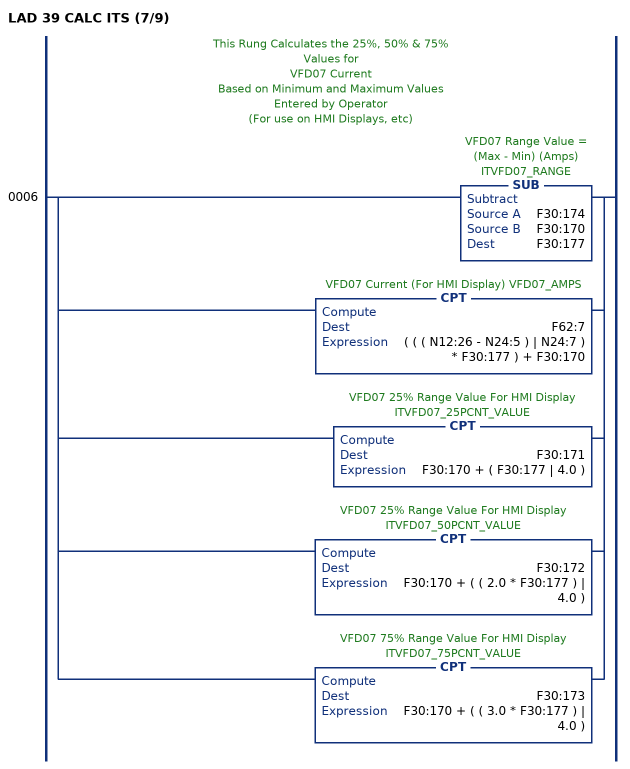
% Rung: 6 %
% This Rung Calculates the 25%, 50% & 75%
% Values for
% VFD07 Current
% Based on Minimum and Maximum Values
% Entered by Operator
% (For use on HMI Displays, etc) %
SOR BST SUB F30:174 F30:170 F30:177 NXB CPT F62:7 " ( ( ( N12:26 - N24:5 ) | N24:7 ) * F30:177 ) + F30:170 " NXB CPT F30:171 " F30:170 + ( F30:177 | 4.0 ) " NXB CPT F30:172 " F30:170 + ( ( 2.0 * F30:177 ) | 4.0 ) " NXB CPT F30:173 " F30:170 + ( ( 3.0 * F30:177 ) | 4.0 ) " BND EOR
%   F30:174  ITVFD07_MAX  "VFD07 Maximum Value (Amps)" %
%   F30:170  ITVFD07_MIN  "VFD07 Minimum Value (Amps)" %
%   F30:177  ITVFD07_RANGE  "VFD07 Range Value = (Max - Min) (Amps)" %
%   F62:7  VFD07_AMPS  "VFD07 Current (For HMI Display)" %
%   N12:26  VFD07_BIN_AMPS  "VFD07 Binary Amps" %
%   N24:5  AI_VOLTAGE_MIN  "Analog Input Minimum Value = 0 VDC (From AI Module)" %
%   N24:7  AI_VOLTAGE_RANGE  "Analog Input Voltage Range Value = (AI_MAX - AI_MIN) For Use Elswhere" %
%   F30:171  ITVFD07_25PCNT_VALUE  "VFD07 25% Range Value For HMI Display" %
%   F30:172  ITVFD07_50PCNT_VALUE  "VFD07 25% Range Value For HMI Display" %
%   F30:173  ITVFD07_75PCNT_VALUE  "VFD07 75% Range Value For HMI Display" %

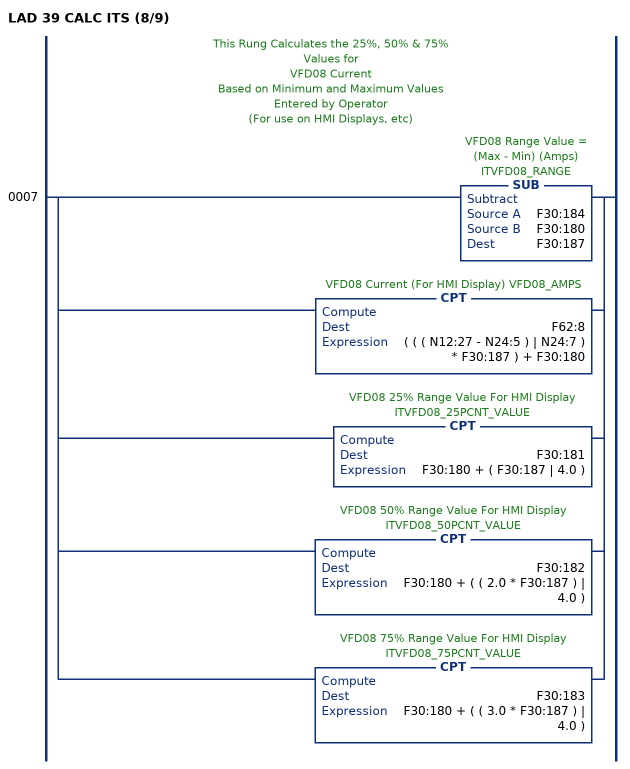
% Rung: 7 %
% This Rung Calculates the 25%, 50% & 75%
% Values for
% VFD08 Current
% Based on Minimum and Maximum Values
% Entered by Operator
% (For use on HMI Displays, etc) %
SOR BST SUB F30:184 F30:180 F30:187 NXB CPT F62:8 " ( ( ( N12:27 - N24:5 ) | N24:7 ) * F30:187 ) + F30:180 " NXB CPT F30:181 " F30:180 + ( F30:187 | 4.0 ) " NXB CPT F30:182 " F30:180 + ( ( 2.0 * F30:187 ) | 4.0 ) " NXB CPT F30:183 " F30:180 + ( ( 3.0 * F30:187 ) | 4.0 ) " BND EOR
%   F30:184  ITVFD08_MAX  "VFD08 Maximum Value (Amps) max = 29.5 ??" %
%   F30:180  ITVFD08_MIN  "VFD08 Minimum Value (Amps)" %
%   F30:187  ITVFD08_RANGE  "VFD08 Range Value = (Max - Min) (Amps)" %
%   F62:8  VFD08_AMPS  "VFD08 Current (For HMI Display)" %
%   N12:27  VFD08_BIN_AMPS  "VFD08 Binary Amps" %
%   N24:5  AI_VOLTAGE_MIN  "Analog Input Minimum Value = 0 VDC (From AI Module)" %
%   N24:7  AI_VOLTAGE_RANGE  "Analog Input Voltage Range Value = (AI_MAX - AI_MIN) For Use Elswhere" %
%   F30:181  ITVFD08_25PCNT_VALUE  "VFD08 25% Range Value For HMI Display" %
%   F30:182  ITVFD08_50PCNT_VALUE  "VFD08 50% Range Value For HMI Display" %
%   F30:183  ITVFD08_75PCNT_VALUE  "VFD08 75% Range Value For HMI Display" %

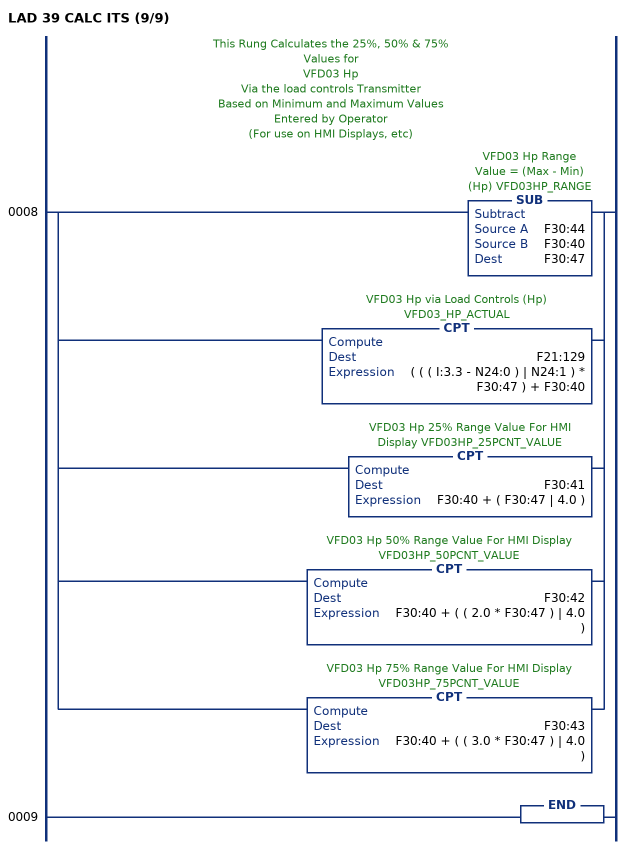
% Rung: 8 %
% This Rung Calculates the 25%, 50% & 75%
% Values for
% VFD03 Hp
% Via the load controls Transmitter
% Based on Minimum and Maximum Values
% Entered by Operator
% (For use on HMI Displays, etc) %
SOR BST SUB F30:44 F30:40 F30:47 NXB CPT F21:129 " ( ( ( I:3.3 - N24:0 ) | N24:1 ) * F30:47 ) + F30:40 " NXB CPT F30:41 " F30:40 + ( F30:47 | 4.0 ) " NXB CPT F30:42 " F30:40 + ( ( 2.0 * F30:47 ) | 4.0 ) " NXB CPT F30:43 " F30:40 + ( ( 3.0 * F30:47 ) | 4.0 ) " BND EOR
%   F30:44  VFD03HP_MAX  "VFD01 Hp Via Load Controls Max (Hp)" %
%   F30:40  VFD03HP_MIN  "VFD01 Hp Via Load Controls Min (Hp)" %
%   F30:47  VFD03HP_RANGE  "VFD03 Hp Range Value = (Max - Min) (Hp)" %
%   F21:129  VFD03_HP_ACTUAL  "VFD03 Hp via Load Controls (Hp)" %
%   I:3.3  VFD03HP_BIN  "VFD03 HP via Load Controls" %
%   N24:0  AI_CURRENT_MIN  "Analog Input Minimum Value = 4 mA DC (From AI Module)" %
%   N24:1  AI_CURRENT_MAX  "Analog Input Maximum Value = 20 mA DC (From AI Module)" %
%   F30:41  VFD03HP_25PCNT_VALUE  "VFD03 Hp 25% Range Value For HMI Display" %
%   F30:42  VFD03HP_50PCNT_VALUE  "VFD03 Hp 50% Range Value For HMI Display" %
%   F30:43  VFD03HP_75PCNT_VALUE  "VFD03 Hp 75% Range Value For HMI Display" %
% Rung: 9 %
SOR END EOR

LADDER 40 "CALC ATS"    % Calculate Densitys from FlowMeters %
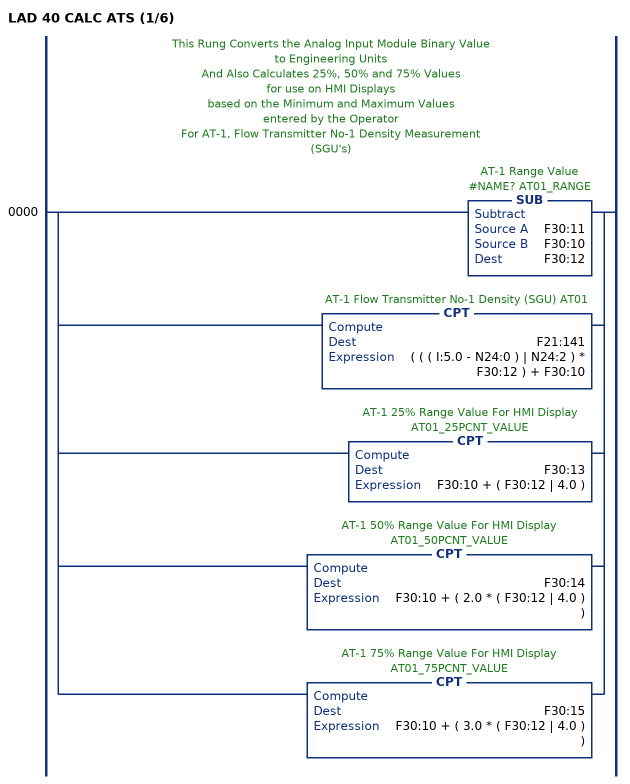
% Rung: 0 %
% This Rung Converts the Analog Input Module Binary Value
% to Engineering Units
% And Also Calculates 25%, 50% and 75% Values
% for use on HMI Displays
% based on the Minimum and Maximum Values
% entered by the Operator
% For AT-1, Flow Transmitter No-1 Density Measurement
% (SGU's) %
SOR BST SUB F30:11 F30:10 F30:12 NXB CPT F21:141 " ( ( ( I:5.0 - N24:0 ) | N24:2 ) * F30:12 ) + F30:10 " NXB CPT F30:13 " F30:10 + ( F30:12 | 4.0 ) " NXB CPT F30:14 " F30:10 + ( 2.0 * ( F30:12 | 4.0 ) ) " NXB CPT F30:15 " F30:10 + ( 3.0 * ( F30:12 | 4.0 ) ) " BND EOR
%   F30:11  AT01_MAX  "AT-1 Maximum Value" %
%   F30:10  AT01_MIN  "AT-1 Minimum Value" %
%   F30:12  AT01_RANGE  "AT-1 Range Value #NAME?" %
%   F21:141  AT01  "AT-1 Flow Transmitter No-1 Density (SGU)" %
%   I:5.0  AT01_BIN  "FT-1 Portable Mass Flowmeter Density Signal No-1" %
%   N24:0  AI_CURRENT_MIN  "Analog Input Minimum Value = 4 mA DC (From AI Module)" %
%   N24:2  AI_CURRENT_RANGE  "Analog Input Current Range Value = (AI_MAX - AI_MIN) For Use Elswhere" %
%   F30:13  AT01_25PCNT_VALUE  "AT-1 25% Range Value For HMI Display" %
%   F30:14  AT01_50PCNT_VALUE  "AT-1 50% Range Value For HMI Display" %
%   F30:15  AT01_75PCNT_VALUE  "AT-1 75% Range Value For HMI Display" %

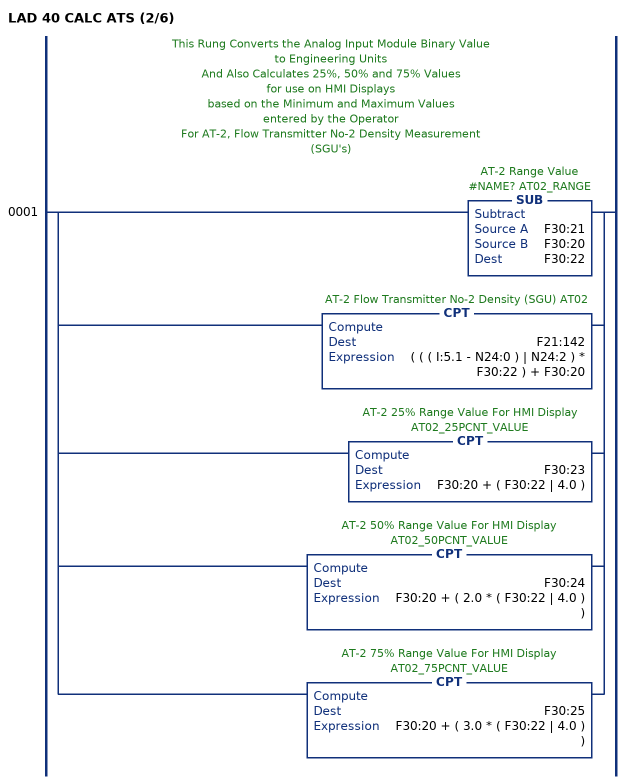
% Rung: 1 %
% This Rung Converts the Analog Input Module Binary Value
% to Engineering Units
% And Also Calculates 25%, 50% and 75% Values
% for use on HMI Displays
% based on the Minimum and Maximum Values
% entered by the Operator
% For AT-2, Flow Transmitter No-2 Density Measurement
% (SGU's) %
SOR BST SUB F30:21 F30:20 F30:22 NXB CPT F21:142 " ( ( ( I:5.1 - N24:0 ) | N24:2 ) * F30:22 ) + F30:20 " NXB CPT F30:23 " F30:20 + ( F30:22 | 4.0 ) " NXB CPT F30:24 " F30:20 + ( 2.0 * ( F30:22 | 4.0 ) ) " NXB CPT F30:25 " F30:20 + ( 3.0 * ( F30:22 | 4.0 ) ) " BND EOR
%   F30:21  AT02_MAX  "AT-2 Maximum Value" %
%   F30:20  AT02_MIN  "AT-2 Minimum Value" %
%   F30:22  AT02_RANGE  "AT-2 Range Value #NAME?" %
%   F21:142  AT02  "AT-2 Flow Transmitter No-2 Density (SGU)" %
%   I:5.1  AT02_BIN  "FT-2 Portable Mass Flowmeter Density Signal No-2" %
%   N24:0  AI_CURRENT_MIN  "Analog Input Minimum Value = 4 mA DC (From AI Module)" %
%   N24:2  AI_CURRENT_RANGE  "Analog Input Current Range Value = (AI_MAX - AI_MIN) For Use Elswhere" %
%   F30:23  AT02_25PCNT_VALUE  "AT-2 25% Range Value For HMI Display" %
%   F30:24  AT02_50PCNT_VALUE  "AT-2 50% Range Value For HMI Display" %
%   F30:25  AT02_75PCNT_VALUE  "AT-2 75% Range Value For HMI Display" %

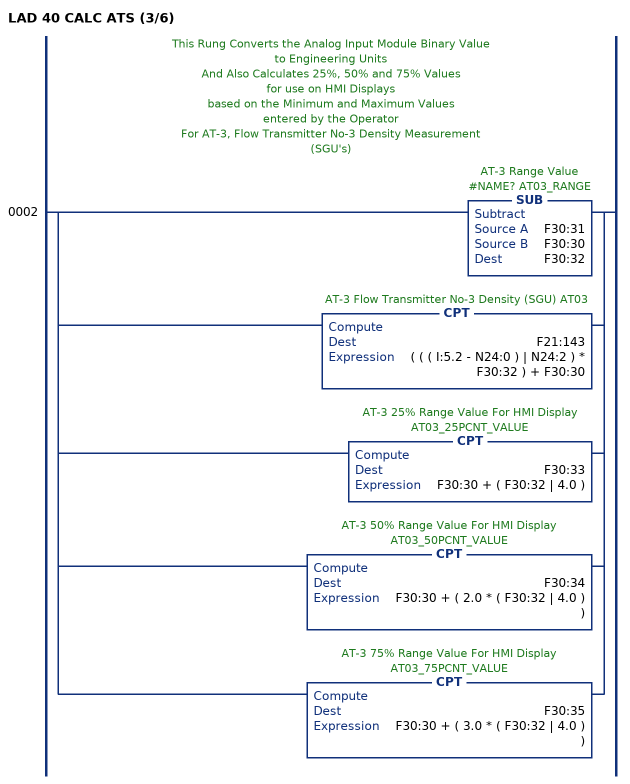
% Rung: 2 %
% This Rung Converts the Analog Input Module Binary Value
% to Engineering Units
% And Also Calculates 25%, 50% and 75% Values
% for use on HMI Displays
% based on the Minimum and Maximum Values
% entered by the Operator
% For AT-3, Flow Transmitter No-3 Density Measurement
% (SGU's) %
SOR BST SUB F30:31 F30:30 F30:32 NXB CPT F21:143 " ( ( ( I:5.2 - N24:0 ) | N24:2 ) * F30:32 ) + F30:30 " NXB CPT F30:33 " F30:30 + ( F30:32 | 4.0 ) " NXB CPT F30:34 " F30:30 + ( 2.0 * ( F30:32 | 4.0 ) ) " NXB CPT F30:35 " F30:30 + ( 3.0 * ( F30:32 | 4.0 ) ) " BND EOR
%   F30:31  AT03_MAX  "AT-3 Maximum Value" %
%   F30:30  AT03_MIN  "AT-3 Minimum Value" %
%   F30:32  AT03_RANGE  "AT-3 Range Value #NAME?" %
%   F21:143  AT03  "AT-3 Flow Transmitter No-3 Density (SGU)" %
%   I:5.2  AT03_BIN  "FT-3 Portable Mass Flowmeter Density Signal No-3" %
%   N24:0  AI_CURRENT_MIN  "Analog Input Minimum Value = 4 mA DC (From AI Module)" %
%   N24:2  AI_CURRENT_RANGE  "Analog Input Current Range Value = (AI_MAX - AI_MIN) For Use Elswhere" %
%   F30:33  AT03_25PCNT_VALUE  "AT-3 25% Range Value For HMI Display" %
%   F30:34  AT03_50PCNT_VALUE  "AT-3 50% Range Value For HMI Display" %
%   F30:35  AT03_75PCNT_VALUE  "AT-3 75% Range Value For HMI Display" %

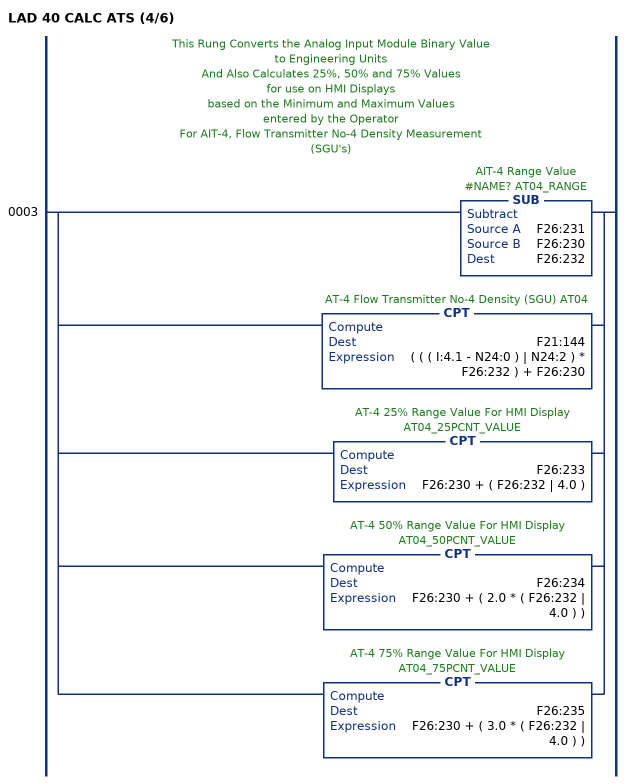
% Rung: 3 %
% This Rung Converts the Analog Input Module Binary Value
% to Engineering Units
% And Also Calculates 25%, 50% and 75% Values
% for use on HMI Displays
% based on the Minimum and Maximum Values
% entered by the Operator
% For AIT-4, Flow Transmitter No-4 Density Measurement
% (SGU's) %
SOR BST SUB F26:231 F26:230 F26:232 NXB CPT F21:144 " ( ( ( I:4.1 - N24:0 ) | N24:2 ) * F26:232 ) + F26:230 " NXB CPT F26:233 " F26:230 + ( F26:232 | 4.0 ) " NXB CPT F26:234 " F26:230 + ( 2.0 * ( F26:232 | 4.0 ) ) " NXB CPT F26:235 " F26:230 + ( 3.0 * ( F26:232 | 4.0 ) ) " BND EOR
%   F26:231  AT04_MAX  "AIT-4 Maximum Value" %
%   F26:230  AT04_MIN  "AIT-4 Minimum Value" %
%   F26:232  AT04_RANGE  "AIT-4 Range Value #NAME?" %
%   F21:144  AT04  "AT-4 Flow Transmitter No-4 Density (SGU)" %
%   I:4.1  AT04_BIN  "FT-4 Portable Mass Flowmeter Density Signal No-4" %
%   N24:0  AI_CURRENT_MIN  "Analog Input Minimum Value = 4 mA DC (From AI Module)" %
%   N24:2  AI_CURRENT_RANGE  "Analog Input Current Range Value = (AI_MAX - AI_MIN) For Use Elswhere" %
%   F26:233  AT04_25PCNT_VALUE  "AT-4 25% Range Value For HMI Display" %
%   F26:234  AT04_50PCNT_VALUE  "AT-4 50% Range Value For HMI Display" %
%   F26:235  AT04_75PCNT_VALUE  "AT-4 75% Range Value For HMI Display" %

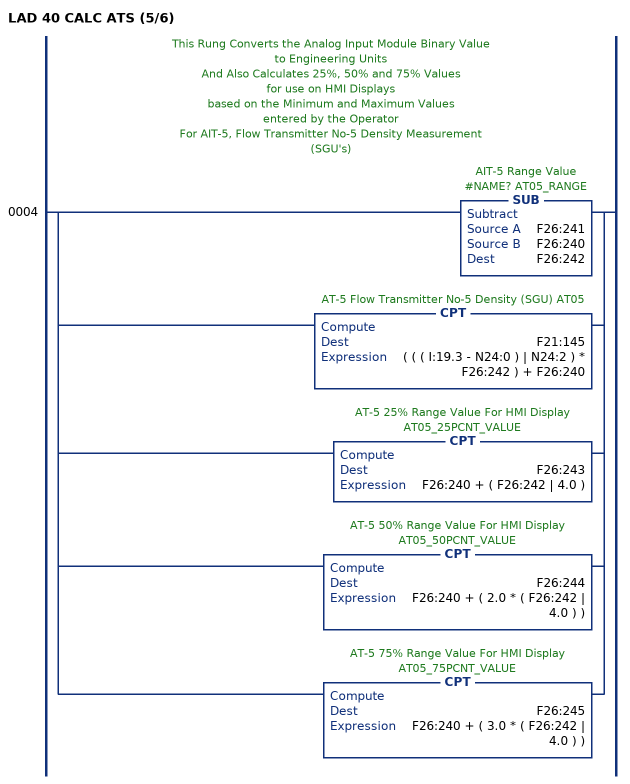
% Rung: 4 %
% This Rung Converts the Analog Input Module Binary Value
% to Engineering Units
% And Also Calculates 25%, 50% and 75% Values
% for use on HMI Displays
% based on the Minimum and Maximum Values
% entered by the Operator
% For AIT-5, Flow Transmitter No-5 Density Measurement
% (SGU's) %
SOR BST SUB F26:241 F26:240 F26:242 NXB CPT F21:145 " ( ( ( I:19.3 - N24:0 ) | N24:2 ) * F26:242 ) + F26:240 " NXB CPT F26:243 " F26:240 + ( F26:242 | 4.0 ) " NXB CPT F26:244 " F26:240 + ( 2.0 * ( F26:242 | 4.0 ) ) " NXB CPT F26:245 " F26:240 + ( 3.0 * ( F26:242 | 4.0 ) ) " BND EOR
%   F26:241  AT05_MAX  "AIT-5 Maximum Value" %
%   F26:240  AT05_MIN  "AIT-5 Minimum Value" %
%   F26:242  AT05_RANGE  "AIT-5 Range Value #NAME?" %
%   F21:145  AT05  "AT-5 Flow Transmitter No-5 Density (SGU)" %
%   I:19.3  AT05_BIN  "FT-5 Portable Mass Flowmeter Density Signal No-5" %
%   N24:0  AI_CURRENT_MIN  "Analog Input Minimum Value = 4 mA DC (From AI Module)" %
%   N24:2  AI_CURRENT_RANGE  "Analog Input Current Range Value = (AI_MAX - AI_MIN) For Use Elswhere" %
%   F26:243  AT05_25PCNT_VALUE  "AT-5 25% Range Value For HMI Display" %
%   F26:244  AT05_50PCNT_VALUE  "AT-5 50% Range Value For HMI Display" %
%   F26:245  AT05_75PCNT_VALUE  "AT-5 75% Range Value For HMI Display" %

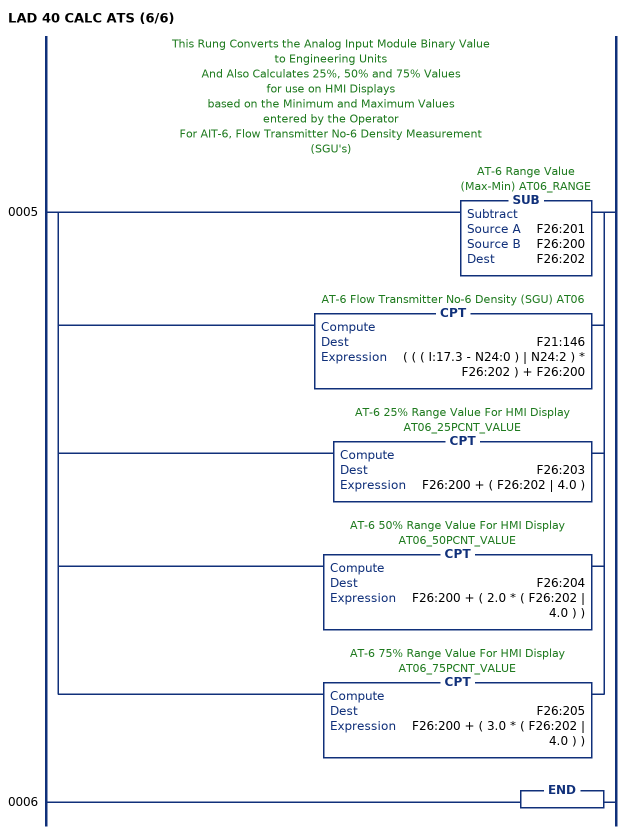
% Rung: 5 %
% This Rung Converts the Analog Input Module Binary Value
% to Engineering Units
% And Also Calculates 25%, 50% and 75% Values
% for use on HMI Displays
% based on the Minimum and Maximum Values
% entered by the Operator
% For AIT-6, Flow Transmitter No-6 Density Measurement
% (SGU's) %
SOR BST SUB F26:201 F26:200 F26:202 NXB CPT F21:146 " ( ( ( I:17.3 - N24:0 ) | N24:2 ) * F26:202 ) + F26:200 " NXB CPT F26:203 " F26:200 + ( F26:202 | 4.0 ) " NXB CPT F26:204 " F26:200 + ( 2.0 * ( F26:202 | 4.0 ) ) " NXB CPT F26:205 " F26:200 + ( 3.0 * ( F26:202 | 4.0 ) ) " BND EOR
%   F26:201  AT06_MAX  "AT-6 Maximum Value" %
%   F26:200  AT06_MIN  "AT-6 Minimum Value" %
%   F26:202  AT06_RANGE  "AT-6 Range Value (Max-Min)" %
%   F21:146  AT06  "AT-6 Flow Transmitter No-6 Density (SGU)" %
%   I:17.3  AT06_BIN  "FT-6 Portable Mass Flowmeter Density Signal No-6" %
%   N24:0  AI_CURRENT_MIN  "Analog Input Minimum Value = 4 mA DC (From AI Module)" %
%   N24:2  AI_CURRENT_RANGE  "Analog Input Current Range Value = (AI_MAX - AI_MIN) For Use Elswhere" %
%   F26:203  AT06_25PCNT_VALUE  "AT-6 25% Range Value For HMI Display" %
%   F26:204  AT06_50PCNT_VALUE  "AT-6 50% Range Value For HMI Display" %
%   F26:205  AT06_75PCNT_VALUE  "AT-6 75% Range Value For HMI Display" %
% Rung: 6 %
SOR END EOR

LADDER 41 "CAL FTAVGS"    % Calculate FT Averages %
